(* PLC project  *)

CONFIGURATION Empty_Module_14
END_CONFIGURATION
